VISUALIZATION InputsScreen  // 2x2
END_VISUALIZATION

(* stored: Version 1.1.0.1, ProductVersion 3.1.4024.13
   Visu InputsScreen: Id {986a406a-4499-44fb-a6b3-c15a724207a3} *)
